// TIA Portal V18 export
FUNCTION "TEMPLATE--v1.0--06_Feedback Error" : Void   // FC7, F_LAD
TITLE = group / bypass contactor feedback errors by I/O Node
{ S7_Optimized_Access := 'TRUE' }
// v1.0 First Emission
BEGIN

REGION Network 1: !!NetworkComment$$
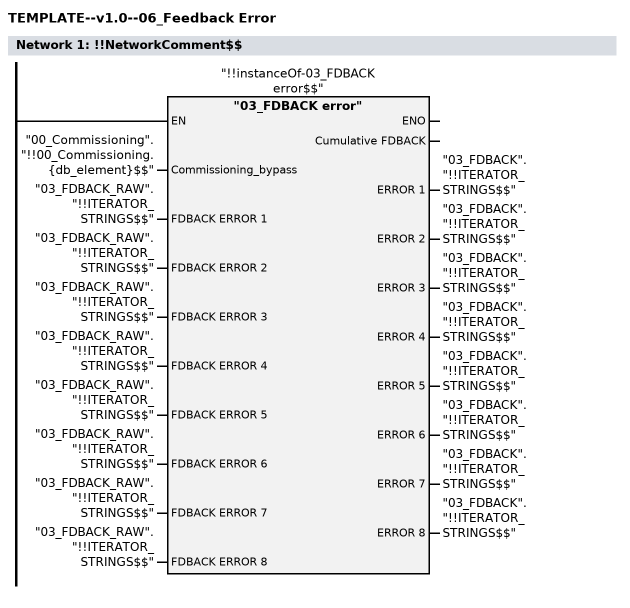
   RUNG wire#powerrail
      "!!instanceOf-03_FDBACK error$$"(Commissioning_bypass := "00_Commissioning"."!!00_Commissioning.{db_element}$$", "FDBACK ERROR 1" := "03_FDBACK_RAW"."!!ITERATOR_STRINGS$$", "FDBACK ERROR 2" := "03_FDBACK_RAW"."!!ITERATOR_STRINGS$$", "FDBACK ERROR 3" := "03_FDBACK_RAW"."!!ITERATOR_STRINGS$$", "FDBACK ERROR 4" := "03_FDBACK_RAW"."!!ITERATOR_STRINGS$$", "FDBACK ERROR 5" := "03_FDBACK_RAW"."!!ITERATOR_STRINGS$$", "FDBACK ERROR 6" := "03_FDBACK_RAW"."!!ITERATOR_STRINGS$$", "FDBACK ERROR 7" := "03_FDBACK_RAW"."!!ITERATOR_STRINGS$$", "FDBACK ERROR 8" := "03_FDBACK_RAW"."!!ITERATOR_STRINGS$$", "Cumulative FDBACK" =>, "ERROR 1" => "03_FDBACK"."!!ITERATOR_STRINGS$$", "ERROR 2" => "03_FDBACK"."!!ITERATOR_STRINGS$$", "ERROR 3" => "03_FDBACK"."!!ITERATOR_STRINGS$$", "ERROR 4" => "03_FDBACK"."!!ITERATOR_STRINGS$$", "ERROR 5" => "03_FDBACK"."!!ITERATOR_STRINGS$$", "ERROR 6" => "03_FDBACK"."!!ITERATOR_STRINGS$$", "ERROR 7" => "03_FDBACK"."!!ITERATOR_STRINGS$$", "ERROR 8" => "03_FDBACK"."!!ITERATOR_STRINGS$$")
   END_RUNG
   // the same network as SCL:
   "!!instanceOf-03_FDBACK error$$"(Commissioning_bypass := "00_Commissioning"."!!00_Commissioning.{db_element}$$",   // "03_FDBACK error"
                           "FDBACK ERROR 1" := "03_FDBACK_RAW"."!!ITERATOR_STRINGS$$",
                           "FDBACK ERROR 2" := "03_FDBACK_RAW"."!!ITERATOR_STRINGS$$",
                           "FDBACK ERROR 3" := "03_FDBACK_RAW"."!!ITERATOR_STRINGS$$",
                           "FDBACK ERROR 4" := "03_FDBACK_RAW"."!!ITERATOR_STRINGS$$",
                           "FDBACK ERROR 5" := "03_FDBACK_RAW"."!!ITERATOR_STRINGS$$",
                           "FDBACK ERROR 6" := "03_FDBACK_RAW"."!!ITERATOR_STRINGS$$",
                           "FDBACK ERROR 7" := "03_FDBACK_RAW"."!!ITERATOR_STRINGS$$",
                           "FDBACK ERROR 8" := "03_FDBACK_RAW"."!!ITERATOR_STRINGS$$",
                           "ERROR 1" => "03_FDBACK"."!!ITERATOR_STRINGS$$",
                           "ERROR 2" => "03_FDBACK"."!!ITERATOR_STRINGS$$",
                           "ERROR 3" => "03_FDBACK"."!!ITERATOR_STRINGS$$",
                           "ERROR 4" => "03_FDBACK"."!!ITERATOR_STRINGS$$",
                           "ERROR 5" => "03_FDBACK"."!!ITERATOR_STRINGS$$",
                           "ERROR 6" => "03_FDBACK"."!!ITERATOR_STRINGS$$",
                           "ERROR 7" => "03_FDBACK"."!!ITERATOR_STRINGS$$",
                           "ERROR 8" => "03_FDBACK"."!!ITERATOR_STRINGS$$");
END_REGION
END_FUNCTION
